Yaskawa INFORM job: X2_50&56B(90_180).JBI

/JOB
//NAME X2_50&56B(90_180)
//POS
///NPOS 378,378,378,17,0,0
///TOOL 0
///POSTYPE PULSE
///PULSE
C00000=-45487,-81749,-76140,-5313,88955,2714
C00001=-100725,-66680,-65098,-5325,101088,-31571
C00002=-135191,-12017,-32267,-15378,118169,-54834
C00003=-185881,43065,27917,-7885,118942,-78845
C00004=-185977,37643,25036,-7838,117929,-78810
C00005=-186017,35528,23980,-7818,117492,-78794
C00006=-186014,35949,26083,-7734,116424,-78717
C00007=-186017,35528,23980,-7818,117492,-78794
C00008=-187441,40927,31967,-8194,115230,-79185
C00009=-186781,38432,29365,-7969,115612,-78957
C00010=-187441,40927,31967,-8194,115230,-79185
C00011=-188109,40448,31416,-8451,115253,-79445
C00012=-188900,38382,29270,-8768,115424,-79764
C00013=-188109,40448,31416,-8451,115253,-79445
C00014=-187906,47991,35532,-8483,116603,-79469
C00015=-135191,-12017,-32267,-15378,118169,-54834
C00016=-100725,-66680,-65098,-5325,101088,-31571
C00017=-68653,-71679,-73408,-24733,95794,-85842
C00018=-66615,-75998,-75470,-24709,95531,-75346
C00019=-80537,-29900,-12555,-12207,96591,-80441
C00020=-81172,-32243,-10721,-12278,94215,-80425
C00021=-81559,-32147,-8308,-12330,92754,-80411
C00022=-81559,-31652,-7175,-12323,92320,-80369
C00023=-79890,-31226,-7999,-11978,93276,-79895
C00024=-78854,-29246,-5136,-11740,92696,-79487
C00025=-78019,-31526,-6644,-11553,92575,-79192
C00026=-78854,-29246,-5136,-11740,92696,-79487
C00027=-78535,-28461,-4244,-11667,92599,-79369
C00028=-79905,-29828,-5160,-11964,92267,-79802
C00029=-78535,-28461,-4244,-11667,92599,-79369
C00030=-80655,-29539,-12313,-12233,96610,-80484
C00031=-172905,9069,10368,-17661,103953,-63205
C00032=-172925,6453,11622,-17490,101927,-62911
C00033=-172953,5852,13232,-17402,100678,-62738
C00034=-172980,6410,14735,-17366,100062,-62659
C00035=-172934,5478,12205,-17429,101103,-62793
C00036=-174868,12262,20269,-17776,99277,-63224
C00037=-175653,10008,18253,-17959,99184,-63493
C00038=-174868,12262,20269,-17776,99277,-63224
C00039=-175466,10534,19114,-17901,98978,-63395
C00040=-174549,8650,17530,-17692,99183,-63095
C00041=-175466,10534,19114,-17901,98978,-63395
C00042=-175364,13912,17144,-18083,101810,-63784
C00043=-143557,-6058,-8183,-20909,99706,-63742
C00044=-116076,-21395,-35361,-8294,99864,41660
C00045=-116170,-16904,-19810,-8141,92666,42104
C00046=-120850,-15711,-13213,-8164,88779,40753
C00047=-120850,-15320,-11697,-8164,88052,40800
C00048=-120850,-15603,-12792,-8164,88575,40767
C00049=-118682,-15547,-12749,-8147,88797,41494
C00050=-118682,-15195,-11396,-8147,88151,41535
C00051=-119909,-15242,-11433,-8154,88024,41123
C00052=-118283,-15171,-11379,-8139,88193,41669
C00053=-118283,-17130,-20118,-8163,92522,41388
C00054=-123081,10517,-9626,-8350,99710,39267
C00055=-134850,49030,33201,-8140,92015,35751
C00056=-141062,59824,58615,-8076,81394,34310
C00057=-142218,64109,67353,-8122,78133,34125
C00058=-142677,66161,71300,-8151,76726,34060
C00059=-142679,67522,74254,-8187,75619,34134
C00060=-142677,66161,71300,-8151,76726,34060
C00061=-139671,63374,68885,-13312,76030,35539
C00062=-140369,64241,69903,-13301,75741,35326
C00063=-139671,63374,68885,-13312,76030,35539
C00064=-139134,61469,65218,-13265,77363,35582
C00065=-137783,55984,53040,-13137,82140,35542
C00066=-137153,72578,74728,-16498,89697,70863
C00067=-137090,72216,76874,-16484,88263,71078
C00068=-137090,73854,80265,-16487,87067,71239
C00069=-137090,73569,79683,-16486,87270,71212
C00070=-137224,70138,75519,-16503,88011,71066
C00071=-137093,72534,77607,-16485,87985,71116
C00072=-140530,75101,78865,-7193,89923,68947
C00073=-141437,70271,73879,-7337,90425,68614
C00074=-141815,70830,74551,-7395,90266,68496
C00075=-141437,68500,69903,-7348,91950,68525
C00076=-138489,28942,16401,-3523,91083,69516
C00077=-135724,-13299,-17509,-11404,84195,25469
C00078=-147110,-27573,-22260,-4915,65599,624
C00079=-144936,-25231,-14401,-13186,59518,1321
C00080=-144776,-24291,-13743,-13234,59620,1373
C00081=-145010,-25647,-14692,-13164,59472,1298
C00082=-145010,-26352,-16893,-13037,60439,1181
C00083=-144720,-24654,-15708,-13123,60625,1273
C00084=-144720,-24280,-14515,-13190,60096,1337
C00085=-145112,-27129,-17933,-12968,60658,1116
C00086=-149472,-33449,-22184,-828,57336,-10794
C00087=-149966,-29456,-16781,-629,56059,-10982
C00088=-150545,-29031,-16493,-385,56096,-11216
C00089=-149966,-29456,-16781,-629,56059,-10982
C00090=-143611,-50009,-41026,-3170,60566,-8561
C00091=-116233,-46088,-51369,-8218,97039,41795
C00092=-133480,-42531,-38521,-8139,89270,36398
C00093=-135471,-40868,-33851,-8115,87069,35859
C00094=-136262,-40121,-31922,-8108,86194,35645
C00095=-136263,-39693,-30384,-8112,85474,35691
C00096=-136262,-40121,-31922,-8108,86194,35645
C00097=-131087,-41226,-31195,-13244,85070,37562
C00098=-132294,-40915,-31003,-13224,84913,37159
C00099=-131087,-41226,-31195,-13244,85070,37562
C00100=-130160,-41921,-33014,-13249,85964,37789
C00101=-127831,-43444,-37404,-13266,88216,38359
C00102=-120126,-54973,-38990,-8175,84580,41274
C00103=-122393,-53255,-34311,-8216,82373,40644
C00104=-123299,-52483,-32378,-8234,81496,40391
C00105=-123299,-51827,-30705,-8247,80810,40437
C00106=-123299,-52483,-32378,-8234,81496,40391
C00107=-117579,-51909,-30953,-13332,81791,42614
C00108=-118939,-51968,-30986,-13356,81559,42167
C00109=-117579,-51909,-30953,-13332,81791,42614
C00110=-116541,-52550,-32737,-13293,82710,42875
C00111=-113955,-53926,-37043,-13200,85024,43525
C00112=-47420,-68852,-70475,-7734,99047,48455
C00113=-58856,-91847,-113443,-3781,117020,74641
C00114=-60236,-59653,-81414,-8514,109210,81552
C00115=-65712,-50088,-67931,-3279,110982,81026
C00116=-65935,-54727,-66929,-3231,107978,81030
C00117=-66231,-56054,-65409,-3227,106352,80970
C00118=-66421,-55660,-64438,-3238,105949,80915
C00119=-66309,-56041,-64890,-3229,106036,80952
C00120=-66048,-59202,-66118,-3188,105179,81066
C00121=-66309,-56041,-64890,-3229,106036,80952
C00122=-65984,-49861,-66477,-3286,110194,80952
C00123=-118683,-89548,-94864,6316,107762,74317
C00124=-118830,-94736,-93309,6169,104171,74077
C00125=-118897,-96147,-91968,6116,102635,73976
C00126=-118911,-94939,-90367,6104,102273,73953
C00127=-118926,-95247,-90740,6105,102345,73951
C00128=-120069,-98591,-91538,5957,101210,73497
C00129=-118926,-95247,-90740,6105,102345,73951
C00130=-124253,-93200,-90530,5582,103647,72150
C00131=-124297,-94887,-90828,5558,102970,72104
C00132=-122332,-96938,-91342,5745,102098,72750
C00133=-124297,-94887,-90828,5558,102970,72104
C00134=-123836,-88068,-93172,5765,107861,72497
C00135=-103947,-87224,-93768,-11726,103256,73456
C00136=-105491,-91629,-91965,-11598,99731,73257
C00137=-106242,-92046,-89539,-11549,97951,73163
C00138=-106280,-91630,-88956,-11545,97803,73164
C00139=-106194,-91849,-89665,-11554,98133,73164
C00140=-106981,-95473,-90615,-11530,96768,73018
C00141=-106194,-91849,-89665,-11554,98133,73164
C00142=-107390,-94613,-90436,-11549,97035,72851
C00143=-105229,-95826,-90624,-11481,96844,73620
C00144=-107390,-94613,-90436,-11549,97035,72851
C00145=-105129,-89034,-93253,-11689,101866,73178
C00146=-117235,-90812,-97794,-11932,101979,68958
C00147=-119184,-94938,-95823,-11777,98434,68628
C00148=-119997,-95229,-93380,-11717,96698,68512
C00149=-120000,-94762,-92745,-11713,96550,68526
C00150=-120085,-95315,-93448,-11717,96683,68484
C00151=-121254,-98780,-94295,-11676,95281,68213
C00152=-120085,-95315,-93448,-11717,96683,68484
C00153=-120732,-97303,-93959,-11694,95897,68335
C00154=-122720,-95241,-93443,-11703,96339,67606
C00155=-120732,-97303,-93959,-11694,95897,68335
C00156=-117928,-92127,-96991,-11873,100734,68840
C00157=-83815,-72409,-71600,-49856,101385,80874
C00158=-86977,-76307,-70966,-49554,98078,81004
C00159=-85918,-79626,-70912,-49280,97499,81857
C00160=-85722,-81512,-70616,-49126,96837,82303
C00161=-87678,-80975,-72090,-49364,96559,81447
C00162=-88529,-80279,-70734,-49348,95782,81419
C00163=-87018,-80378,-72384,-49396,97246,81423
C00164=-92255,-82689,-76075,-49623,95110,79856
C00165=-92255,-82357,-74554,-49552,94603,80124
C00166=-91886,-84274,-76762,-49584,95051,80076
C00167=-87038,-78982,-77882,-49995,99948,79968
C00168=-111885,-94745,-96836,-21175,93099,57761
C00169=-115356,-96241,-94167,-20812,89966,57066
C00170=-116782,-95898,-92034,-20669,88542,56800
C00171=-116805,-94979,-90810,-20667,88272,56838
C00172=-117687,-92490,-90484,-20584,89063,56388
C00173=-119638,-92586,-90524,-20383,88555,55777
C00174=-116782,-95072,-90979,-20669,88331,56836
C00175=-116675,-98914,-91892,-20684,87033,57096
C00176=-116782,-95072,-90979,-20669,88331,56836
C00177=-111949,-93327,-94846,-21154,92619,57823
C00178=-55380,-134082,-104834,-55812,75253,81172
C00179=-61753,-134169,-102482,-55825,70609,80463
C00180=-64815,-132350,-99998,-55791,68452,80067
C00181=-65073,-131468,-99170,-55790,68267,80036
C00182=-65012,-131683,-99347,-55795,68302,80050
C00183=-67421,-134585,-100123,-55949,66292,79958
C00184=-65012,-131683,-99347,-55795,68302,80050
C00185=-66833,-133758,-99865,-55902,66793,79972
C00186=-68699,-130981,-99713,-55278,66469,79035
C00187=-66833,-133758,-99865,-55902,66793,79972
C00188=-57706,-134492,-103408,-55942,73242,81128
C00189=-64785,-112873,-118243,-24954,102118,81978
C00190=-94326,-86621,-83484,35338,109503,87169
C00191=-91634,-91881,-83017,35113,105930,87131
C00192=-90294,-93871,-83332,35163,104694,87298
C00193=-90673,-91662,-79967,34941,104076,86932
C00194=-96279,-95614,-77654,39133,100534,74699
C00195=-97530,-94207,-78400,39125,102027,74707
C00196=-99906,-89889,-79610,39309,105429,74936
C00197=-93707,-90060,-101982,2678,109676,68403
C00198=-85859,-88563,-85007,-37375,108858,60120
C00199=-89767,-92929,-84612,-37372,105169,59726
C00200=-92261,-92553,-83552,-37602,103718,59151
C00201=-87809,-89294,-77804,-36664,104133,60948
C00202=-97825,-97090,-85633,-28728,98264,58810
C00203=-105101,-94972,-90460,-21721,102166,53461
C00204=-101619,-91841,-92201,-21697,105576,54126
C00205=-110011,-90138,-98551,-28023,73725,47627
C00206=-114073,-86949,-94757,-26595,71811,46539
C00207=-115644,-85550,-93357,-26007,71199,46082
C00208=-116827,-38850,-76508,-24575,105038,42322
C00209=-113194,-138803,-104651,-24561,74823,49786
C00210=-115995,-123992,-100550,-21546,88254,42562
C00211=-113813,-124047,-101616,-21486,89414,43150
C00212=-108993,-124666,-104884,-21332,92253,44397
C00213=-109211,-98340,-98499,-17204,97884,65653
C00214=-111963,-101539,-96259,-17038,94417,65168
C00215=-114319,-101452,-95162,-16976,93323,64488
C00216=-121130,-95827,-93982,-7505,98794,69297
C00217=-120137,-94785,-95042,-7509,100063,69562
C00218=-118600,-90390,-96949,-7580,103607,69872
C00219=-87744,-101201,-89183,-32285,100120,63549
C00220=-91822,-104522,-87796,-32421,96378,62986
C00221=-93007,-105888,-87219,-32449,95024,62902
C00222=-125171,-100001,-94421,-10746,96250,68519
C00223=-112189,-112791,-97117,-10082,92847,73286
C00224=-125737,-104595,-94231,-123,98676,80328
C00225=-125012,-83838,-85262,-564,111182,80520
C00226=-124880,-77934,-85992,-554,114665,80551
C00227=-118378,-61430,-80227,500,113656,60542
C00228=-119635,-65792,-78782,346,110532,60082
C00229=-120344,-67374,-78220,265,109375,59827
C00230=-117636,-69991,-79065,562,108539,60782
C00231=-61499,-79673,-75485,5801,99043,80116
C00232=-59682,-78713,-74784,5933,98973,80740
C00233=-58729,-76685,-75165,6027,100171,81128
C00234=-59096,-71470,-86943,6341,110071,81508
C00235=-60236,-59653,-81414,-8514,109210,81552
C00236=-58856,-91847,-113443,-3781,117020,74641
C00237=-47420,-68852,-70475,-7734,99047,48455
C00238=-126000,-95797,-97639,7032,71909,-3420
C00239=-125334,-73481,-62420,7403,61720,-3825
C00240=-136814,-5072,7481,-118,87452,-82611
C00241=-137691,-48649,-34753,-2434,90887,-80546
C00242=-137775,-50281,-31902,-2439,88294,-80524
C00243=-137810,-50839,-30689,-2442,87260,-80516
C00244=-135168,-51719,-31185,-2214,87179,-79626
C00245=-133081,-52293,-31505,-2034,87136,-78923
C00246=-130377,-52882,-31830,-1800,87108,-78013
C00247=-130424,-52342,-33062,-1804,88142,-78044
C00248=-109921,-30503,-12357,-16555,100596,-88828
C00249=-109696,-31149,-11049,-16422,99550,-88604
C00250=-109235,-30430,-9939,-16278,99338,-88414
C00251=-108888,-29584,-8170,-16145,98777,-88217
C00252=-108084,-28000,-11018,-16080,101404,-88284
C00253=-146524,-12798,-32,1632,107432,-69723
C00254=-145636,-15796,-268,1931,106019,-69429
C00255=-148965,-15940,435,4110,105287,-67260
C00256=-149102,-15441,1522,4054,104879,-67319
C00257=-149548,-12799,1040,3936,106552,-67422
C00258=-137932,-46455,-34045,-2456,91570,-80642
C00259=-130584,-47998,-33152,-21701,103265,-82699
C00260=-131924,-51228,-32028,-21814,100720,-82725
C00261=-132035,-52540,-31560,-21763,99795,-82595
C00262=-133096,-52283,-31444,-22032,99580,-82945
C00263=-135164,-51769,-31262,-22544,99165,-83631
C00264=-135522,-51681,-31234,-22630,99088,-83749
C00265=-135156,-50442,-31749,-22619,100068,-83801
C00266=-145953,-54402,-37679,-17502,96627,-81619
C00267=-150690,-47590,-28968,-15173,97194,-77528
C00268=-141688,-67515,-39498,-21463,83995,-90539
C00269=-138380,-68197,-47605,-21119,89179,-90269
C00270=-135468,-61779,-51499,-19715,96090,-83313
C00271=-146504,11659,2252,-17659,107540,-74925
C00272=-144153,-20650,-13732,-15502,93070,1402
C00273=-144800,-23297,881,-19511,75808,35743
C00274=-150190,-18698,6871,-14781,74684,33485
C00275=-147156,-18843,9866,-19821,72199,35502
C00276=-149144,-27907,3634,-19922,70959,34997
C00277=-146448,7715,36431,-22348,89479,40067
C00278=-145889,24730,54854,-22060,94685,42086
C00279=-143819,24834,51946,-21414,96917,42392
C00280=-152079,-13657,11289,-11329,66320,30599
C00281=-154288,-10621,16286,-8724,64794,29674
C00282=-151904,106,24911,-8978,65250,30498
C00283=-150907,-2622,20158,-8985,66862,30731
C00284=-148148,-14759,14441,-17311,62501,33163
C00285=-153240,-11311,16162,-10073,64214,30249
C00286=-151074,-2242,23117,-10293,64850,30978
C00287=-150611,-3939,19670,-10247,66139,31030
C00288=-148132,-4021,18992,-11949,66408,32059
C00289=-147374,-3194,21269,-13667,65169,32648
C00290=-146197,4054,27436,-13805,65293,33065
C00291=-152653,-4647,20265,-5226,59206,14792
C00292=-154418,-25114,11432,-1101,38258,22446
C00293=-154596,-31771,2822,-953,40134,22334
C00294=-135242,-54877,-19518,-11584,43472,31405
C00295=-131236,-19596,-17600,-13529,71052,30429
C00296=-140706,-23702,-4175,-12836,48543,13474
C00297=-139806,-19028,764,-13410,48067,13944
C00298=-142658,-11173,6654,-18063,50404,18129
C00299=-141158,-15186,3600,-18761,50563,18771
C00300=-142435,-9097,12555,-18853,48016,18701
C00301=-142049,-7157,14085,-20669,49065,20425
C00302=-142257,-9387,11148,-20387,49635,20204
C00303=-144365,-13616,3568,-3735,54240,8270
C00304=-145823,-13393,6250,-1324,50480,7579
C00305=-145532,-11229,7851,-5107,50939,11169
C00306=-140850,-20387,-3678,-6927,53662,12969
C00307=-124087,52798,66602,-30516,90034,63653
C00308=-125471,40650,54753,-32699,86509,59979
C00309=-125334,44720,63004,-32764,84027,60751
C00310=-121896,62283,77480,-32170,85396,61678
C00311=-136105,75569,91402,-14378,82982,62392
C00312=-137341,77557,93952,-14596,82241,62066
C00313=-141168,85934,104737,-15299,79317,61146
C00314=-141539,87094,106260,-15375,78917,61072
C00315=-141741,86606,105619,-15400,79023,60993
C00316=-141171,84118,98448,-15196,82155,60793
C00317=-132001,54931,46945,-19188,86263,30068
C00318=-132148,77644,76370,-19381,80137,30989
C00319=-133367,86129,89618,-16102,76593,30820
C00320=-134153,81899,83498,-14098,78199,30187
C00321=-134623,67905,67625,-12481,69763,30818
C00322=-134986,36263,31606,-9687,63888,24183
C00323=-134666,27103,16729,-9479,68314,23935
C00324=-130420,39472,29702,-18859,92900,38190
C00325=-131547,40725,34135,-18850,90663,38133
C00326=-134032,43651,38469,-15292,90000,37322
C00327=-134717,31522,25950,-15335,91293,36921
C00328=-133273,44284,38720,-16717,93907,38368
C00329=-131769,55424,45596,-17778,98765,39318
C00330=-127656,48680,32292,-16283,104912,42086
C00331=-116663,7338,4481,-17873,88938,41861
C00332=-82713,25471,38030,-41323,96034,53690
C00333=-86390,18515,43854,-41800,88900,54935
C00334=-85131,26101,60384,-49314,87065,55858
C00335=-88537,53193,89669,-50569,82685,56609
C00336=-87361,53333,88208,-50128,83897,56499
C00337=-87606,32039,49279,-49923,92343,51642
C00338=-120401,-109118,-96895,-24846,84275,3219
C00339=-171543,-75667,-77525,32488,107850,-47798
C00340=-132158,4506,-3799,21442,87877,-38180
C00341=-135903,57798,67571,35925,99624,-57782
C00342=-135834,61045,74411,35664,97518,-58450
C00343=-136852,65101,79345,35223,97458,-58869
C00344=-135824,2781,6571,30163,84476,-36889
C00345=-132310,1940,5711,27060,83090,-36079
C00346=-131484,15794,17971,27055,82441,-35917
C00347=-137267,10911,1717,27131,91031,-36122
C00348=-146203,-27363,-23504,26744,90214,-39705
C00349=-126939,-13199,-3011,17863,102554,-59788
C00350=-123418,-15871,2353,18433,97326,-59310
C00351=-121180,-11626,8848,18695,97500,-62472
C00352=-121861,-10835,10563,18474,97032,-62783
C00353=-122570,-10261,12471,18233,96354,-63137
C00354=-117580,-17478,3718,13074,93264,-62869
C00355=-122301,-18046,-869,17501,95215,-65467
C00356=-137808,-17234,-5965,14129,101643,-70132
C00357=-160865,-72571,-62696,26432,95765,-43985
C00358=-33343,-40499,-55087,-21473,103101,-25780
C00359=-34531,-11607,-34091,-29923,106513,-58273
C00360=-34985,-14035,-31998,-29527,104140,-57811
C00361=-34859,-13066,-29764,-29400,103418,-57570
C00362=-36609,-20544,-36296,-27578,100646,-57392
C00363=-52934,-69115,-66821,-23349,86237,-60131
C00364=-53727,-71032,-72534,-20342,85587,-60124
C00365=-146487,-18846,-10598,-19725,94468,-68028
C00366=-155890,-2777,10204,-12003,101739,-63000
C00367=-156750,-807,13372,-12200,100693,-63202
C00368=-157443,816,16029,-12357,99805,-63356
C00369=-157211,1579,14506,-12356,101141,-63409
C00370=-145375,-16597,89,-21780,91791,-76946
C00371=-153197,-12711,3322,-13630,93085,-80939
C00372=-151754,-15041,1558,-14681,91924,-82917
C00373=-145475,-7318,12723,-24819,92922,-88907
C00374=-142776,-6009,11285,-24301,95132,-88379
C00375=-137963,-3619,4000,-23654,101759,-87941
C00376=-103503,-37411,-26995,-22689,104461,-77175
C00377=2000,-113393,-91320,0,88983,0
BC00000=213492,669309,586749
BC00001=279836,668491,248946
BC00002=347085,719558,248946
BC00003=397217,757626,248946
BC00004=397217,757626,248946
BC00005=397217,757626,248946
BC00006=397217,757626,248946
BC00007=397217,757626,248946
BC00008=397217,757626,248946
BC00009=397217,757626,248946
BC00010=397217,757626,248946
BC00011=397217,757626,248946
BC00012=397217,757626,248946
BC00013=397217,757626,248946
BC00014=397217,757626,248946
BC00015=347085,719558,248946
BC00016=279836,668491,248946
BC00017=74259,666735,420956
BC00018=74259,755070,420956
BC00019=74259,755070,420956
BC00020=74259,755070,420956
BC00021=74259,755070,420956
BC00022=74259,755070,420956
BC00023=74259,755070,420956
BC00024=74259,755070,420956
BC00025=74259,755070,420956
BC00026=74259,755070,420956
BC00027=74259,755070,420956
BC00028=74259,755070,420956
BC00029=74259,755070,420956
BC00030=74259,755070,420956
BC00031=168853,756619,369390
BC00032=168853,756619,369390
BC00033=168853,756619,369390
BC00034=168853,756619,369390
BC00035=168853,756619,369390
BC00036=168853,756619,369390
BC00037=168853,756619,369390
BC00038=168853,756619,369390
BC00039=168853,756619,369390
BC00040=168853,756619,369390
BC00041=168853,756619,369390
BC00042=168853,756619,369390
BC00043=153069,767391,383312
BC00044=133900,791089,347452
BC00045=133902,791088,347446
BC00046=133902,791088,347446
BC00047=133902,791088,347446
BC00048=133902,791088,347446
BC00049=133902,791088,347446
BC00050=133902,791088,347446
BC00051=133902,791088,347446
BC00052=133902,791088,347446
BC00053=133902,791088,347446
BC00054=133900,791089,347452
BC00055=133900,791089,347452
BC00056=133900,791089,347452
BC00057=133900,791089,347452
BC00058=133900,791089,347452
BC00059=133900,791089,347452
BC00060=133900,791089,347452
BC00061=133900,791089,347452
BC00062=133900,791089,347452
BC00063=133900,791089,347452
BC00064=133900,791089,347452
BC00065=133900,791089,347452
BC00066=133900,791089,347451
BC00067=133900,791089,347451
BC00068=133900,791089,347451
BC00069=133900,791089,347451
BC00070=133900,791089,347451
BC00071=133900,791089,347451
BC00072=133900,791089,347451
BC00073=133900,791089,347451
BC00074=133900,791089,347451
BC00075=133900,791089,347451
BC00076=133900,791089,347451
BC00077=133900,791089,347451
BC00078=133899,791089,347449
BC00079=133899,791089,347449
BC00080=133899,791089,347449
BC00081=133899,791089,347449
BC00082=133899,791089,347449
BC00083=133899,791089,347449
BC00084=133899,791089,347449
BC00085=133899,791089,347449
BC00086=133899,791089,347449
BC00087=133899,791089,347449
BC00088=133899,791089,347449
BC00089=133899,791089,347449
BC00090=133899,791089,347449
BC00091=91689,791089,305907
BC00092=91689,791089,305907
BC00093=91689,791089,305907
BC00094=91689,791089,305907
BC00095=91689,791089,305907
BC00096=91689,791089,305907
BC00097=91689,791089,305907
BC00098=91689,791089,305907
BC00099=91689,791089,305907
BC00100=91689,791089,305907
BC00101=91689,791089,305907
BC00102=65725,737951,350532
BC00103=65725,737951,350532
BC00104=65725,737951,350532
BC00105=65725,737951,350532
BC00106=65725,737951,350532
BC00107=65725,737951,350532
BC00108=65725,737951,350532
BC00109=65725,737951,350532
BC00110=65725,737951,350532
BC00111=65725,737951,350532
BC00112=45615,670175,524343
BC00113=269563,738996,1075229
BC00114=398174,782420,1075175
BC00115=398174,782420,1075175
BC00116=398174,782420,1075175
BC00117=398174,782420,1075175
BC00118=398174,782420,1075175
BC00119=398174,782420,1075175
BC00120=398174,782420,1075175
BC00121=398174,782420,1075175
BC00122=398174,782420,1075175
BC00123=387355,830302,1075175
BC00124=387355,830302,1075175
BC00125=387355,830302,1075175
BC00126=387355,830302,1075175
BC00127=387355,830302,1075175
BC00128=387355,830302,1075175
BC00129=387355,830302,1075175
BC00130=387355,830302,1075175
BC00131=387355,830302,1075175
BC00132=387355,830302,1075175
BC00133=387355,830302,1075175
BC00134=387355,830302,1075175
BC00135=398174,816751,1075175
BC00136=398174,816751,1075175
BC00137=398174,816751,1075175
BC00138=398174,816751,1075175
BC00139=398174,816751,1075175
BC00140=398174,816751,1075175
BC00141=398174,816751,1075175
BC00142=398174,816751,1075175
BC00143=398174,816751,1075175
BC00144=398174,816751,1075175
BC00145=398174,816751,1075175
BC00146=394174,829691,1075175
BC00147=394174,829691,1075175
BC00148=394174,829691,1075175
BC00149=394174,829691,1075175
BC00150=394174,829691,1075175
BC00151=394174,829691,1075175
BC00152=394174,829691,1075175
BC00153=394174,829691,1075175
BC00154=394174,829691,1075175
BC00155=394174,829691,1075175
BC00156=394174,829691,1075175
BC00157=398174,810220,1075175
BC00158=398174,810220,1075175
BC00159=398174,810220,1075175
BC00160=398174,810220,1075175
BC00161=398174,810220,1075175
BC00162=398174,810220,1075175
BC00163=398174,810220,1075175
BC00164=398174,810220,1075175
BC00165=398174,810220,1075175
BC00166=398174,810220,1075175
BC00167=398174,810220,1075175
BC00168=398174,820048,1075175
BC00169=398174,820048,1075175
BC00170=398174,820048,1075175
BC00171=398174,820048,1075175
BC00172=398174,820048,1075175
BC00173=398174,820048,1075175
BC00174=398174,820048,1075175
BC00175=398174,820048,1075175
BC00176=398174,820048,1075175
BC00177=398174,820048,1075175
BC00178=357533,882194,1075175
BC00179=357533,882194,1075175
BC00180=357533,882194,1075175
BC00181=357533,882194,1075175
BC00182=357533,882194,1075175
BC00183=357533,882194,1075175
BC00184=357533,882194,1075175
BC00185=357533,882194,1075175
BC00186=357533,882194,1075175
BC00187=357533,882194,1075175
BC00188=357533,882194,1075175
BC00189=340885,876696,1075175
BC00190=309760,866417,1075175
BC00191=309760,866417,1075175
BC00192=309760,866417,1075175
BC00193=309760,866417,1075175
BC00194=309760,866417,1075175
BC00195=309760,866417,1075175
BC00196=309760,866417,1075175
BC00197=346143,852026,1075175
BC00198=394169,833030,1075175
BC00199=394169,833030,1075175
BC00200=394169,833030,1075175
BC00201=394169,833030,1075175
BC00202=394169,833030,1075175
BC00203=394169,833030,1075175
BC00204=394169,833030,1075175
BC00205=398174,851161,1075175
BC00206=398174,851161,1075175
BC00207=398174,851161,1075175
BC00208=398174,851161,1075175
BC00209=398174,851161,1075175
BC00210=398174,851161,1075175
BC00211=398174,851161,1075175
BC00212=398174,851161,1075175
BC00213=383646,835540,1075175
BC00214=383646,835540,1075175
BC00215=383647,835541,1075174
BC00216=383646,835540,1075175
BC00217=383646,835540,1075175
BC00218=383646,835540,1075175
BC00219=398174,834635,1075175
BC00220=398174,834635,1075175
BC00221=398174,834635,1075175
BC00222=398174,834635,1075175
BC00223=398174,834635,1075175
BC00224=398174,834635,1075175
BC00225=398174,834635,1075175
BC00226=398174,834635,1075175
BC00227=398174,805809,1075175
BC00228=398174,805809,1075175
BC00229=398174,805809,1075175
BC00230=398174,805809,1075175
BC00231=398174,805809,1075175
BC00232=398174,805809,1075175
BC00233=398174,805809,1075175
BC00234=398174,805809,1075175
BC00235=398174,782420,1075175
BC00236=269563,738996,1075229
BC00237=45615,670175,524343
BC00238=94279,678895,315353
BC00239=94279,729713,315353
BC00240=135603,767285,503004
BC00241=127958,749365,374153
BC00242=127958,749365,374153
BC00243=127958,749365,374153
BC00244=127958,749365,374153
BC00245=127958,749365,374153
BC00246=127958,749365,374153
BC00247=127958,749365,374153
BC00248=127958,749365,374153
BC00249=127958,749365,374153
BC00250=127958,749365,374153
BC00251=127958,749365,374153
BC00252=127958,749365,374153
BC00253=127958,749365,374153
BC00254=127958,749365,374153
BC00255=127958,749365,374153
BC00256=127958,749365,374153
BC00257=127958,749365,374153
BC00258=127958,749365,374153
BC00259=104823,777232,320967
BC00260=104823,777232,320967
BC00261=104823,777232,320967
BC00262=104823,777232,320967
BC00263=104823,777232,320967
BC00264=104823,777232,320967
BC00265=104823,777232,320967
BC00266=104823,777232,320967
BC00267=104823,777232,320967
BC00268=104823,777232,320967
BC00269=104823,777232,320967
BC00270=104823,777232,320967
BC00271=148105,732999,367459
BC00272=136799,735677,423222
BC00273=131883,736842,447466
BC00274=131883,736842,447466
BC00275=131883,736842,447466
BC00276=131883,736842,447466
BC00277=131883,736842,447466
BC00278=131883,736842,447466
BC00279=131883,736842,447466
BC00280=135864,729332,463750
BC00281=135864,729332,463750
BC00282=135864,729332,463750
BC00283=135864,729332,463750
BC00284=135957,757580,463073
BC00285=135957,757580,463073
BC00286=135957,757580,463073
BC00287=135957,757580,463073
BC00288=132965,771777,450481
BC00289=132965,771777,450481
BC00290=132965,771777,450481
BC00291=132965,771777,450481
BC00292=132965,771777,450481
BC00293=132965,771777,450481
BC00294=132965,771777,450481
BC00295=129716,779092,399778
BC00296=129716,779092,399778
BC00297=129716,779092,399778
BC00298=129716,779092,399778
BC00299=129716,779092,399778
BC00300=129716,779092,399778
BC00301=129716,779092,399778
BC00302=129716,779092,399778
BC00303=129716,779092,399778
BC00304=129716,779092,399778
BC00305=129716,779092,399778
BC00306=129716,779092,399778
BC00307=129716,795131,399778
BC00308=129716,795131,399778
BC00309=129716,795131,399778
BC00310=129716,795131,399778
BC00311=129716,795131,399778
BC00312=129716,795131,399778
BC00313=129716,795131,399778
BC00314=129716,795131,399778
BC00315=129716,795131,399778
BC00316=129716,795131,399778
BC00317=124387,791089,316625
BC00318=124387,789553,316625
BC00319=119293,789553,296084
BC00320=117256,789553,287867
BC00321=117256,789553,287867
BC00322=112196,789553,268708
BC00323=112196,789553,268708
BC00324=113936,791089,281332
BC00325=113936,791089,281332
BC00326=113936,791089,281332
BC00327=113936,791089,281332
BC00328=113936,791089,281332
BC00329=113936,791089,281332
BC00330=113936,791089,281332
BC00331=116869,773103,397669
BC00332=116869,773103,397669
BC00333=116869,773103,397669
BC00334=116869,773103,397669
BC00335=116869,773103,397669
BC00336=116869,773103,397669
BC00337=116996,772325,398387
BC00338=133980,668182,494562
BC00339=6392,668182,323571
BC00340=6392,776369,323571
BC00341=6392,786149,323571
BC00342=6392,786149,323571
BC00343=6392,786149,323571
BC00344=6392,786149,323571
BC00345=6392,786149,323571
BC00346=6392,786149,323571
BC00347=6392,786149,323571
BC00348=6392,734041,397800
BC00349=6392,734041,397800
BC00350=6392,734041,397800
BC00351=5812,733225,400788
BC00352=6392,733053,399870
BC00353=6392,734041,402294
BC00354=6392,734041,399183
BC00355=6392,734041,397800
BC00356=6392,734041,397800
BC00357=6392,674729,482291
BC00358=159586,688686,294802
BC00359=173113,745279,189268
BC00360=173113,745279,189268
BC00361=173113,745279,189268
BC00362=173113,745279,189268
BC00363=173113,745279,189268
BC00364=173113,745279,189268
BC00365=329544,744159,387532
BC00366=329544,744159,387532
BC00367=329544,744159,387532
BC00368=329544,744159,387532
BC00369=329544,744159,387532
BC00370=329544,744159,387532
BC00371=329544,744159,387532
BC00372=329544,744159,387532
BC00373=329544,744159,387532
BC00374=329544,744159,387532
BC00375=329544,744159,387532
BC00376=296372,673105,416449
BC00377=87189,666204,1075229
EC00000=798156,1112951
EC00001=798156,1112951
EC00002=798156,1112951
EC00003=798156,1112951
EC00004=798156,1112951
EC00005=798156,1112951
EC00006=798156,1112951
EC00007=798156,1112951
EC00008=798156,1112951
EC00009=798156,1112951
EC00010=798156,1112951
EC00011=798156,1112951
EC00012=798156,1112951
EC00013=798156,1112951
EC00014=798156,1112951
EC00015=798156,1112951
EC00016=798156,1112951
EC00017=798156,1112951
EC00018=798156,1112951
EC00019=798156,1112951
EC00020=798156,1112951
EC00021=798156,1112951
EC00022=798156,1112951
EC00023=798156,1112951
EC00024=798156,1112951
EC00025=798156,1112951
EC00026=798156,1112951
EC00027=798156,1112951
EC00028=798156,1112951
EC00029=798156,1112951
EC00030=798156,1112951
EC00031=798156,1112951
EC00032=798156,1112951
EC00033=798156,1112951
EC00034=798156,1112951
EC00035=798156,1112951
EC00036=798156,1112951
EC00037=798156,1112951
EC00038=798156,1112951
EC00039=798156,1112951
EC00040=798156,1112951
EC00041=798156,1112951
EC00042=798156,1112951
EC00043=798156,1112951
EC00044=798156,1112951
EC00045=798154,1112949
EC00046=798154,1112949
EC00047=798154,1112949
EC00048=798154,1112949
EC00049=798154,1112949
EC00050=798154,1112949
EC00051=798154,1112949
EC00052=798154,1112949
EC00053=798154,1112949
EC00054=798156,1112951
EC00055=798156,1112951
EC00056=798156,1112951
EC00057=798156,1112951
EC00058=798156,1112951
EC00059=798156,1112951
EC00060=798156,1112951
EC00061=798156,1112951
EC00062=798156,1112951
EC00063=798156,1112951
EC00064=798156,1112951
EC00065=798156,1112951
EC00066=798155,1112949
EC00067=798155,1112949
EC00068=798155,1112949
EC00069=798155,1112949
EC00070=798155,1112949
EC00071=798155,1112949
EC00072=798155,1112949
EC00073=798155,1112949
EC00074=798155,1112949
EC00075=798155,1112949
EC00076=798155,1112949
EC00077=798155,1112949
EC00078=798154,1112948
EC00079=798154,1112948
EC00080=798154,1112948
EC00081=798154,1112948
EC00082=798154,1112948
EC00083=798154,1112948
EC00084=798154,1112948
EC00085=798154,1112948
EC00086=798154,1112948
EC00087=798154,1112948
EC00088=798154,1112948
EC00089=798154,1112948
EC00090=798154,1112948
EC00091=798156,1112951
EC00092=798156,1112951
EC00093=798156,1112951
EC00094=798156,1112951
EC00095=798156,1112951
EC00096=798156,1112951
EC00097=798156,1112951
EC00098=798156,1112951
EC00099=798156,1112951
EC00100=798156,1112951
EC00101=798156,1112951
EC00102=798156,1112951
EC00103=798156,1112951
EC00104=798156,1112951
EC00105=798156,1112951
EC00106=798156,1112951
EC00107=798156,1112951
EC00108=798156,1112951
EC00109=798156,1112951
EC00110=798156,1112951
EC00111=798156,1112951
EC00112=798156,1112951
EC00113=906908,1112951
EC00114=975524,1112951
EC00115=975524,1112951
EC00116=975524,1112951
EC00117=975524,1112951
EC00118=975524,1112951
EC00119=975524,1112951
EC00120=975524,1112951
EC00121=975524,1112951
EC00122=975524,1112951
EC00123=975524,1112951
EC00124=975524,1112951
EC00125=975524,1112951
EC00126=975524,1112951
EC00127=975524,1112951
EC00128=975524,1112951
EC00129=975524,1112951
EC00130=975524,1112951
EC00131=975524,1112951
EC00132=975524,1112951
EC00133=975524,1112951
EC00134=975524,1112951
EC00135=975524,1112951
EC00136=975524,1112951
EC00137=975524,1112951
EC00138=975524,1112951
EC00139=975524,1112951
EC00140=975524,1112951
EC00141=975524,1112951
EC00142=975524,1112951
EC00143=975524,1112951
EC00144=975524,1112951
EC00145=975524,1112951
EC00146=975524,1112951
EC00147=975524,1112951
EC00148=975524,1112951
EC00149=975524,1112951
EC00150=975524,1112951
EC00151=975524,1112951
EC00152=975524,1112951
EC00153=975524,1112951
EC00154=975524,1112951
EC00155=975524,1112951
EC00156=975524,1112951
EC00157=975524,1112951
EC00158=975524,1112951
EC00159=975524,1112951
EC00160=975524,1112951
EC00161=975524,1112951
EC00162=975524,1112951
EC00163=975524,1112951
EC00164=975524,1112951
EC00165=975524,1112951
EC00166=975524,1112951
EC00167=975524,1112951
EC00168=975524,1112951
EC00169=975524,1112951
EC00170=975524,1112951
EC00171=975524,1112951
EC00172=975524,1112951
EC00173=975524,1112951
EC00174=975524,1112951
EC00175=975524,1112951
EC00176=975524,1112951
EC00177=975524,1112951
EC00178=975524,1112951
EC00179=975524,1112951
EC00180=975524,1112951
EC00181=975524,1112951
EC00182=975524,1112951
EC00183=975524,1112951
EC00184=975524,1112951
EC00185=975524,1112951
EC00186=975524,1112951
EC00187=975524,1112951
EC00188=975524,1112951
EC00189=975524,1112951
EC00190=975524,1112951
EC00191=975524,1112951
EC00192=975524,1112951
EC00193=975524,1112951
EC00194=975524,1112951
EC00195=975524,1112951
EC00196=975524,1112951
EC00197=975524,1112951
EC00198=975524,1112951
EC00199=975524,1112951
EC00200=975524,1112951
EC00201=975524,1112951
EC00202=975524,1112951
EC00203=975524,1112951
EC00204=975524,1112951
EC00205=975524,1112951
EC00206=975524,1112951
EC00207=975524,1112951
EC00208=975524,1112951
EC00209=975524,1112951
EC00210=975524,1112951
EC00211=975524,1112951
EC00212=975524,1112951
EC00213=975524,1112951
EC00214=975524,1112951
EC00215=975522,1112950
EC00216=975524,1112951
EC00217=975524,1112951
EC00218=975524,1112951
EC00219=975524,1112951
EC00220=975524,1112951
EC00221=975524,1112951
EC00222=975524,1112951
EC00223=975524,1112951
EC00224=975524,1112951
EC00225=975524,1112951
EC00226=975524,1112951
EC00227=975524,1112951
EC00228=975524,1112951
EC00229=975524,1112951
EC00230=975524,1112951
EC00231=975524,1112951
EC00232=975524,1112951
EC00233=975524,1112951
EC00234=975524,1112951
EC00235=975524,1112951
EC00236=906908,1112951
EC00237=798156,1112951
EC00238=798156,1112951
EC00239=798156,1112951
EC00240=798156,1112951
EC00241=798156,1112951
EC00242=798156,1112951
EC00243=798156,1112951
EC00244=798156,1112951
EC00245=798156,1112951
EC00246=798156,1112951
EC00247=798156,1112951
EC00248=798156,1112951
EC00249=798156,1112951
EC00250=798156,1112951
EC00251=798156,1112951
EC00252=798156,1112951
EC00253=798156,1112951
EC00254=798156,1112951
EC00255=798156,1112951
EC00256=798156,1112951
EC00257=798156,1112951
EC00258=798156,1112951
EC00259=798156,1112951
EC00260=798156,1112951
EC00261=798156,1112951
EC00262=798156,1112951
EC00263=798156,1112951
EC00264=798156,1112951
EC00265=798156,1112951
EC00266=798156,1112951
EC00267=798156,1112951
EC00268=798156,1112951
EC00269=798156,1112951
EC00270=798156,1112951
EC00271=798156,1112951
EC00272=798156,1112951
EC00273=798156,1112951
EC00274=798156,1112951
EC00275=798156,1112951
EC00276=798156,1112951
EC00277=798156,1112951
EC00278=798156,1112951
EC00279=798156,1112951
EC00280=798156,1112951
EC00281=798156,1112951
EC00282=798156,1112951
EC00283=798156,1112951
EC00284=798156,1112951
EC00285=798156,1112951
EC00286=798156,1112951
EC00287=798156,1112951
EC00288=798156,1112951
EC00289=798156,1112951
EC00290=798156,1112951
EC00291=798156,1112951
EC00292=798156,1112951
EC00293=798156,1112951
EC00294=798156,1112951
EC00295=798156,1112951
EC00296=798156,1112951
EC00297=798156,1112951
EC00298=798156,1112951
EC00299=798156,1112951
EC00300=798156,1112951
EC00301=798156,1112951
EC00302=798156,1112951
EC00303=798156,1112951
EC00304=798156,1112951
EC00305=798156,1112951
EC00306=798156,1112951
EC00307=798156,1112951
EC00308=798156,1112951
EC00309=798156,1112951
EC00310=798156,1112951
EC00311=798156,1112951
EC00312=798156,1112951
EC00313=798156,1112951
EC00314=798156,1112951
EC00315=798156,1112951
EC00316=798156,1112951
EC00317=798156,1112951
EC00318=798156,1112951
EC00319=798156,1112951
EC00320=798156,1112951
EC00321=798156,1112951
EC00322=798156,1112951
EC00323=798156,1112951
EC00324=798156,1112951
EC00325=798156,1112951
EC00326=798156,1112951
EC00327=798156,1112951
EC00328=798156,1112951
EC00329=798156,1112951
EC00330=798156,1112951
EC00331=798156,1112951
EC00332=798156,1112951
EC00333=798156,1112951
EC00334=798156,1112951
EC00335=798156,1112951
EC00336=798156,1112951
EC00337=798156,1112951
EC00338=798156,1112951
EC00339=798156,1112951
EC00340=798156,1112951
EC00341=798156,1112951
EC00342=798156,1112951
EC00343=798156,1112951
EC00344=798156,1112951
EC00345=798156,1112951
EC00346=798156,1112951
EC00347=798156,1112951
EC00348=798156,1112951
EC00349=798156,1112951
EC00350=798156,1112951
EC00351=798156,1112951
EC00352=798156,1112951
EC00353=798156,1112951
EC00354=798156,1112951
EC00355=798156,1112951
EC00356=798156,1112951
EC00357=798156,1112951
EC00358=798156,1112951
EC00359=798156,1112951
EC00360=798156,1112951
EC00361=798156,1112951
EC00362=798156,1112951
EC00363=798156,1112951
EC00364=798156,1112951
EC00365=798156,1112951
EC00366=798156,1112951
EC00367=798156,1112951
EC00368=798156,1112951
EC00369=798156,1112951
EC00370=798156,1112951
EC00371=798156,1112951
EC00372=798156,1112951
EC00373=798156,1112951
EC00374=798156,1112951
EC00375=798156,1112951
EC00376=798156,1112951
EC00377=798156,1112951
///POSTYPE BASE
///RECTAN
///RCONF 0,0,0,0,0,0,0,0,0,0,0,0,0,0,0,0,0,0,0,0,0,0,0,0
P00006=0.222,-3.123,-1.508,0.0000,0.0000,0.0000
P00021=-0.225,-6.128,-0.405,0.0000,0.0000,0.0000
P00022=0.222,-3.123,-1.508,0.0000,0.0000,0.0000
P00023=0.143,-0.036,0.682,0.0000,0.0000,0.0000
P00024=0.145,-0.552,1.326,0.0000,0.0000,0.0000
P00025=-2.003,0.006,0.728,0.0000,0.0000,0.0000
P00026=0.562,-0.002,-0.337,0.0000,0.0000,0.0000
P00027=-0.746,0.015,-9.096,0.0000,0.0000,0.0000
P00028=-2.237,-0.018,-7.702,0.0000,0.0000,0.0000
P00029=-2.156,-0.086,-4.681,0.0000,0.0000,0.0000
P00032=1.957,0.503,-7.217,0.0000,0.0000,0.0000
///RCONF 0,0,0,0,1,0,0,0,0,0,0,0,0,0,0,0,0,0,0,0,0,0,0,0
P00033=-0.123,0.612,-5.012,0.0000,0.0000,0.0000
///RCONF 0,0,0,0,0,0,0,0,0,0,0,0,0,0,0,0,0,0,0,0,0,0,0,0
P00034=-0.304,0.773,-2.693,0.0000,0.0000,0.0000
P00050=4.296,-4.501,-0.826,0.0000,0.0000,0.0000
P00051=0.367,3.892,0.009,0.0000,0.0000,0.0000
P00063=0.036,-0.654,-3.005,0.0000,0.0000,0.0000
P00099=-0.837,6.343,-3.499,0.0000,0.0000,0.0000
//INST
///DATE 2024/11/05 10:16
///ATTR SC,RW
///GROUP1 RB1,BS1
///GROUP2 ST1
NOP
'X2_50&56B(90_180)
'Down
MOVJ C00000 BC00000 VJ=100.00  +MOVJ EC00000 VJ=100.00
MOVJ C00001 BC00001 VJ=100.00  +MOVJ EC00001 VJ=100.00
MOVJ C00002 BC00002 VJ=100.00  +MOVJ EC00002 VJ=100.00
'Path S4514
SFTOF3D
MOVJ C00003 BC00003 VJ=100.00  +MOVJ EC00003 VJ=100.00
MOVL C00004 BC00004 V=800.0  +MOVJ EC00004 VJ=100.00
SMOVL C00005 BC00005 V=166.7  +MOVJ EC00005
SREFP 3 C00006 BC00006  +REFP EC00006
CALL JOB:SEARCH-R1-S13D
SET P034 P006
SFTON3D P034
SMOVL C00007 BC00007 V=166.7  +MOVJ EC00007
SMOVL C00008 BC00008 V=166.7  +MOVJ EC00008
SREFP 3 C00009 BC00009  +REFP EC00009
CALL JOB:SEARCH-R1-S13D
SET P034 P006
SFTON3D P034
SMOVL C00010 BC00010 V=166.7  +MOVJ EC00010
SMOVL C00011 BC00011 V=166.7  +MOVJ EC00011
SREFP 3 C00012 BC00012  +REFP EC00012
CALL JOB:SEARCH-R1-S13D
SET P034 P006
SFTON3D P034
SMOVL C00013 BC00013 V=166.7  +MOVJ EC00013
MOVL C00014 BC00014 V=1000.0  +MOVJ EC00014 VJ=100.00
'EndPath S4514
MOVJ C00015 BC00015 VJ=100.00  +MOVJ EC00015 VJ=100.00
MOVJ C00016 BC00016 VJ=100.00  +MOVJ EC00016 VJ=100.00
MOVJ C00017 BC00017 VJ=100.00  +MOVJ EC00017 VJ=100.00
MOVJ C00018 BC00018 VJ=100.00  +MOVJ EC00018 VJ=100.00
'Path S4515
SFTOF3D
MOVJ C00019 BC00019 VJ=100.00  +MOVJ EC00019 VJ=100.00
MOVL C00020 BC00020 V=800.0  +MOVJ EC00020 VJ=100.00
SMOVL C00021 BC00021 V=166.7  +MOVJ EC00021
SREFP 3 C00022 BC00022  +REFP EC00022
CALL JOB:SEARCH-R1-S13D
SET P033 P006
SFTON3D P033
SMOVL C00023 BC00023 V=250.0  +MOVJ EC00023
SMOVL C00024 BC00024 V=166.7  +MOVJ EC00024
SREFP 3 C00025 BC00025  +REFP EC00025
CALL JOB:SEARCH-R1-S13D
SET P033 P006
SFTON3D P033
SMOVL C00026 BC00026 V=166.7  +MOVJ EC00026
SMOVL C00027 BC00027 V=166.7  +MOVJ EC00027
SREFP 3 C00028 BC00028  +REFP EC00028
CALL JOB:SEARCH-R1-S13D
SET P033 P006
SFTON3D P033
SMOVL C00029 BC00029 V=166.7  +MOVJ EC00029
MOVL C00030 BC00030 V=1000.0  +MOVJ EC00030 VJ=100.00
'EndPath S4515
'Path S4516
SFTOF3D
MOVJ C00031 BC00031 VJ=100.00  +MOVJ EC00031 VJ=100.00
MOVL C00032 BC00032 V=800.0  +MOVJ EC00032 VJ=100.00
SMOVL C00033 BC00033 V=166.7  +MOVJ EC00033
SREFP 3 C00034 BC00034  +REFP EC00034
CALL JOB:SEARCH-R1-S13D
SET P032 P006
SFTON3D P032
SMOVL C00035 BC00035 V=166.7  +MOVJ EC00035
SMOVL C00036 BC00036 V=166.7  +MOVJ EC00036
SREFP 3 C00037 BC00037  +REFP EC00037
CALL JOB:SEARCH-R1-S13D
SET P032 P006
SFTON3D P032
SMOVL C00038 BC00038 V=166.7  +MOVJ EC00038
SMOVL C00039 BC00039 V=166.7  +MOVJ EC00039
SREFP 3 C00040 BC00040  +REFP EC00040
CALL JOB:SEARCH-R1-S13D
SET P032 P006
SFTON3D P032
SMOVL C00041 BC00041 V=166.7  +MOVJ EC00041
MOVL C00042 BC00042 V=1000.0  +MOVJ EC00042 VJ=100.00
'EndPath S4516
MOVJ C00043 BC00043 VJ=100.00  +MOVJ EC00043 VJ=100.00
MOVJ C00044 BC00044 VJ=100.00  +MOVJ EC00044 VJ=100.00
MOVL C00045 BC00045 V=800.0  +MOVJ EC00045 VJ=100.00
SMOVL C00046 BC00046 V=250.0  +MOVJ EC00046
SREFP 3 C00047 BC00047  +REFP EC00047
CALL JOB:SEARCH-R1-S13D
SET P099 P006
SFTON3D P099
SMOVL C00048 BC00048 V=166.7  +MOVJ EC00048
SMOVL C00049 BC00049 V=250.0  +MOVJ EC00049
SMOVL C00050 BC00050 V=166.7  +MOVJ EC00050
SREFP 3 C00051 BC00051  +REFP EC00051
CALL JOB:SEARCH-R1-S13D
SET P099 P006
SFTON3D P099
SMOVL C00052 BC00052 V=166.7  +MOVJ EC00052
SMOVL C00053 BC00053 V=800.0  +MOVJ EC00053
SFTOF3D
MOVJ C00054 BC00054 VJ=100.00  +MOVJ EC00054 VJ=100.00
'Path S4517
SFTOF3D
MOVJ C00055 BC00055 VJ=100.00  +MOVJ EC00055 VJ=100.00
'Path S4519
SFTOF3D
MOVJ C00056 BC00056 VJ=100.00  +MOVJ EC00056 VJ=100.00
MOVL C00057 BC00057 V=800.0  +MOVJ EC00057 VJ=100.00
SMOVL C00058 BC00058 V=166.7  +MOVJ EC00058
SREFP 3 C00059 BC00059  +REFP EC00059
CALL JOB:SEARCH-R1-S13D
SET P029 P006
SFTON3D P029
SMOVL C00060 BC00060 V=166.7  +MOVJ EC00060
SMOVL C00061 BC00061 V=166.7  +MOVJ EC00061
SREFP 3 C00062 BC00062  +REFP EC00062
CALL JOB:SEARCH-R1-S13D
SET P029 P006
SFTON3D P029
SMOVL C00063 BC00063 V=166.7  +MOVJ EC00063
SFTOF3D
MOVL C00064 BC00064 V=800.0  +MOVJ EC00064 VJ=100.00
MOVL C00065 BC00065 V=1000.0  +MOVJ EC00065 VJ=100.00
SMOVL C00066 BC00066 V=250.0  +MOVJ EC00066
SMOVL C00067 BC00067 V=250.0  +MOVJ EC00067
SREFP 3 C00068 BC00068  +REFP EC00068
CALL JOB:SEARCH-R1-S13D
SET P050 P006
SFTON3D P050
SMOVL C00069 BC00069 V=166.7  +MOVJ EC00069
SREFP 3 C00070 BC00070  +REFP EC00070
CALL JOB:SEARCH-R1-S13D
SET P050 P006
SFTON3D P050
SMOVL C00071 BC00071 V=166.7  +MOVJ EC00071
SMOVL C00072 BC00072 V=250.0  +MOVJ EC00072
SMOVL C00073 BC00073 V=250.0  +MOVJ EC00073
SREFP 3 C00074 BC00074  +REFP EC00074
CALL JOB:SEARCH-R1-S13D
SET P050 P006
SFTON3D P050
SMOVL C00075 BC00075 V=166.7  +MOVJ EC00075
SFTOF3D
SMOVL C00076 BC00076 V=666.7  +MOVJ EC00076
SMOVL C00077 BC00077 V=666.7  +MOVJ EC00077
SMOVL C00078 BC00078 V=250.0  +MOVJ EC00078
SMOVL C00079 BC00079 V=250.0  +MOVJ EC00079
SREFP 3 C00080 BC00080  +REFP EC00080
CALL JOB:SEARCH-R1-S13D
SET P051 P006
SFTON3D P051
SMOVL C00081 BC00081 V=166.7  +MOVJ EC00081
SMOVL C00082 BC00082 V=250.0  +MOVJ EC00082
SMOVL C00083 BC00083 V=133.3  +MOVJ EC00083
SREFP 3 C00084 BC00084  +REFP EC00084
CALL JOB:SEARCH-R1-S13D
SET P051 P006
SFTON3D P051
SMOVL C00085 BC00085 V=250.0  +MOVJ EC00085
SMOVL C00086 BC00086 V=500.0  +MOVJ EC00086
SMOVL C00087 BC00087 V=250.0  +MOVJ EC00087
SREFP 3 C00088 BC00088  +REFP EC00088
CALL JOB:SEARCH-R1-S13D
SET P051 P006
SFTON3D P051
SMOVL C00089 BC00089 V=166.7  +MOVJ EC00089
SFTOF3D
SMOVL C00090 BC00090 V=666.7  +MOVJ EC00090
'EndPath S4519
MOVJ C00091 BC00091 VJ=100.00  +MOVJ EC00091 VJ=100.00
'Path S4520
SFTOF3D
MOVJ C00092 BC00092 VJ=100.00  +MOVJ EC00092 VJ=100.00
MOVL C00093 BC00093 V=800.0  +MOVJ EC00093 VJ=100.00
SMOVL C00094 BC00094 V=133.3  +MOVJ EC00094
SREFP 3 C00095 BC00095  +REFP EC00095
CALL JOB:SEARCH-R1-S13D
SET P028 P006
SFTON3D P028
SMOVL C00096 BC00096 V=166.7  +MOVJ EC00096
SMOVL C00097 BC00097 V=166.7  +MOVJ EC00097
SREFP 3 C00098 BC00098  +REFP EC00098
CALL JOB:SEARCH-R1-S13D
SET P028 P006
SFTON3D P028
SMOVL C00099 BC00099 V=166.7  +MOVJ EC00099
MOVL C00100 BC00100 V=800.0  +MOVJ EC00100 VJ=100.00
MOVL C00101 BC00101 V=1000.0  +MOVJ EC00101 VJ=100.00
'EndPath S4520
'Path S4521
SFTOF3D
MOVJ C00102 BC00102 VJ=100.00  +MOVJ EC00102 VJ=100.00
MOVL C00103 BC00103 V=800.0  +MOVJ EC00103 VJ=100.00
SMOVL C00104 BC00104 V=166.7  +MOVJ EC00104
SREFP 3 C00105 BC00105  +REFP EC00105
CALL JOB:SEARCH-R1-S13D
SET P027 P006
SFTON3D P027
SMOVL C00106 BC00106 V=166.7  +MOVJ EC00106
SMOVL C00107 BC00107 V=166.7  +MOVJ EC00107
SREFP 3 C00108 BC00108  +REFP EC00108
CALL JOB:SEARCH-R1-S13D
SET P027 P006
SFTON3D P027
SMOVL C00109 BC00109 V=166.7  +MOVJ EC00109
MOVL C00110 BC00110 V=800.0  +MOVJ EC00110 VJ=100.00
MOVL C00111 BC00111 V=1000.0  +MOVJ EC00111 VJ=100.00
'EndPath S4521
MOVJ C00112 BC00112 VJ=100.00  +MOVJ EC00112 VJ=100.00
'Up
MOVJ C00113 BC00113 VJ=100.00  +MOVJ EC00113 VJ=100.00
MOVJ C00114 BC00114 VJ=100.00  +MOVJ EC00114 VJ=100.00
'Path S4522
SFTOF3D
MOVJ C00115 BC00115 VJ=100.00  +MOVJ EC00115 VJ=100.00
MOVL C00116 BC00116 V=800.0  +MOVJ EC00116 VJ=100.00
SMOVL C00117 BC00117 V=166.7  +MOVJ EC00117
SREFP 3 C00118 BC00118  +REFP EC00118
CALL JOB:SEARCH-R1-S13D
SET P026 P006
SFTON3D P026
SMOVL C00119 BC00119 V=166.7  +MOVJ EC00119
SREFP 3 C00120 BC00120  +REFP EC00120
CALL JOB:SEARCH-R1-S13D
SET P026 P006
SFTON3D P026
SMOVL C00121 BC00121 V=166.7  +MOVJ EC00121
MOVL C00122 BC00122 V=1000.0  +MOVJ EC00122 VJ=100.00
'EndPath S4522
'Path S4523
SFTOF3D
MOVJ C00123 BC00123 VJ=100.00  +MOVJ EC00123 VJ=100.00
MOVL C00124 BC00124 V=800.0  +MOVJ EC00124 VJ=100.00
SMOVL C00125 BC00125 V=166.7  +MOVJ EC00125
SREFP 3 C00126 BC00126  +REFP EC00126
CALL JOB:SEARCH-R1-S13D
SET P025 P006
SFTON3D P025
SMOVL C00127 BC00127 V=166.7  +MOVJ EC00127
SREFP 3 C00128 BC00128  +REFP EC00128
CALL JOB:SEARCH-R1-S13D
SET P025 P006
SFTON3D P025
SMOVL C00129 BC00129 V=166.7  +MOVJ EC00129
SMOVL C00130 BC00130 V=166.7  +MOVJ EC00130
SMOVL C00131 BC00131 V=166.7  +MOVJ EC00131
SREFP 3 C00132 BC00132  +REFP EC00132
CALL JOB:SEARCH-R1-S13D
SET P025 P006
SFTON3D P025
SMOVL C00133 BC00133 V=166.7  +MOVJ EC00133
MOVL C00134 BC00134 V=1000.0  +MOVJ EC00134 VJ=100.00
'EndPath S4523
'Path S4524
SFTOF3D
MOVJ C00135 BC00135 VJ=100.00  +MOVJ EC00135 VJ=100.00
MOVL C00136 BC00136 V=800.0  +MOVJ EC00136 VJ=100.00
SMOVL C00137 BC00137 V=166.7  +MOVJ EC00137
SREFP 3 C00138 BC00138  +REFP EC00138
CALL JOB:SEARCH-R1-S13D
SET P024 P006
SFTON3D P024
SMOVL C00139 BC00139 V=166.7  +MOVJ EC00139
SREFP 3 C00140 BC00140  +REFP EC00140
CALL JOB:SEARCH-R1-S13D
SET P024 P006
SFTON3D P024
SMOVL C00141 BC00141 V=166.7  +MOVJ EC00141
SMOVL C00142 BC00142 V=166.7  +MOVJ EC00142
SREFP 3 C00143 BC00143  +REFP EC00143
CALL JOB:SEARCH-R1-S13D
SET P024 P006
SFTON3D P024
SMOVL C00144 BC00144 V=166.7  +MOVJ EC00144
MOVL C00145 BC00145 V=1000.0  +MOVJ EC00145 VJ=100.00
'EndPath S4524
'Path S4525
SFTOF3D
MOVJ C00146 BC00146 VJ=100.00  +MOVJ EC00146 VJ=100.00
MOVL C00147 BC00147 V=800.0  +MOVJ EC00147 VJ=100.00
SMOVL C00148 BC00148 V=166.7  +MOVJ EC00148
SREFP 3 C00149 BC00149  +REFP EC00149
CALL JOB:SEARCH-R1-S13D
SET P023 P006
SFTON3D P023
SMOVL C00150 BC00150 V=166.7  +MOVJ EC00150
SREFP 3 C00151 BC00151  +REFP EC00151
CALL JOB:SEARCH-R1-S13D
SET P023 P006
SFTON3D P023
SMOVL C00152 BC00152 V=166.7  +MOVJ EC00152
SMOVL C00153 BC00153 V=166.7  +MOVJ EC00153
SREFP 3 C00154 BC00154  +REFP EC00154
CALL JOB:SEARCH-R1-S13D
SET P023 P006
SFTON3D P023
SMOVL C00155 BC00155 V=166.7  +MOVJ EC00155
MOVL C00156 BC00156 V=1000.0  +MOVJ EC00156 VJ=100.00
'EndPath S4525
'Path S4729
SFTOF3D
MOVJ C00157 BC00157 VJ=100.00  +MOVJ EC00157 VJ=100.00
MOVL C00158 BC00158 V=800.0  +MOVJ EC00158 VJ=100.00
SMOVL C00159 BC00159 V=166.7  +MOVJ EC00159
SREFP 3 C00160 BC00160  +REFP EC00160
CALL JOB:SEARCH-R1-S13D
SET P063 P006
SFTON3D P063
SMOVL C00161 BC00161 V=166.7  +MOVJ EC00161
SREFP 3 C00162 BC00162  +REFP EC00162
CALL JOB:SEARCH-R1-S13D
SET P063 P006
SFTON3D P063
SMOVL C00163 BC00163 V=166.7  +MOVJ EC00163
SMOVL C00164 BC00164 V=166.7  +MOVJ EC00164
SREFP 3 C00165 BC00165  +REFP EC00165
CALL JOB:SEARCH-R1-S13D
SET P063 P006
SFTON3D P063
SMOVL C00166 BC00166 V=166.7  +MOVJ EC00166
MOVL C00167 BC00167 V=1000.0  +MOVJ EC00167 VJ=100.00
'EndPath S4729
'Path S4526
SFTOF3D
MOVJ C00168 BC00168 VJ=100.00  +MOVJ EC00168 VJ=100.00
MOVL C00169 BC00169 V=800.0  +MOVJ EC00169 VJ=100.00
SMOVL C00170 BC00170 V=166.7  +MOVJ EC00170
SREFP 3 C00171 BC00171  +REFP EC00171
CALL JOB:SEARCH-R1-S13D
SET P022 P006
SFTON3D P022
SMOVL C00172 BC00172 V=166.7  +MOVJ EC00172
SREFP 3 C00173 BC00173  +REFP EC00173
CALL JOB:SEARCH-R1-S13D
SET P022 P006
SFTON3D P022
SMOVL C00174 BC00174 V=166.7  +MOVJ EC00174
SREFP 3 C00175 BC00175  +REFP EC00175
CALL JOB:SEARCH-R1-S13D
SET P022 P006
SFTON3D P022
SMOVL C00176 BC00176 V=166.7  +MOVJ EC00176
MOVL C00177 BC00177 V=1000.0  +MOVJ EC00177 VJ=100.00
'EndPath S4526
'Path S4527
SFTOF3D
MOVJ C00178 BC00178 VJ=100.00  +MOVJ EC00178 VJ=100.00
MOVL C00179 BC00179 V=800.0  +MOVJ EC00179 VJ=100.00
SMOVL C00180 BC00180 V=166.7  +MOVJ EC00180
SREFP 3 C00181 BC00181  +REFP EC00181
CALL JOB:SEARCH-R1-S13D
SET P021 P006
SFTON3D P021
SMOVL C00182 BC00182 V=166.7  +MOVJ EC00182
SREFP 3 C00183 BC00183  +REFP EC00183
CALL JOB:SEARCH-R1-S13D
SET P021 P006
SFTON3D P021
SMOVL C00184 BC00184 V=250.0  +MOVJ EC00184
SMOVL C00185 BC00185 V=166.7  +MOVJ EC00185
SREFP 3 C00186 BC00186  +REFP EC00186
CALL JOB:SEARCH-R1-S13D
SET P021 P006
SFTON3D P021
SMOVL C00187 BC00187 V=166.7  +MOVJ EC00187
MOVL C00188 BC00188 V=1000.0  +MOVJ EC00188 VJ=100.00
'EndPath S4527
MOVJ C00189 BC00189 VJ=100.00  +MOVJ EC00189 VJ=100.00
'Path W4730
SFTOF3D
SFTON3D P024
MOVJ C00190 BC00190 VJ=100.00  +MOVJ EC00190 VJ=100.00
SMOVL C00191 BC00191 V=800.0  +MOVJ EC00191
SMOVL C00192 BC00192 V=150.0 PL=0  +MOVJ EC00192
MACRO1 MJ#(0) ARGF14
ARCON
SMOVL C00193 BC00193 V=10.0  +MOVJ EC00193
SMOVL C00194 BC00194 V=11.7  +MOVJ EC00194
ARCOF
SMOVL C00195 BC00195 V=800.0  +MOVJ EC00195
SMOVL C00196 BC00196 V=1000.0  +MOVJ EC00196
SFTOF3D
'EndPath W4730
MOVJ C00197 BC00197 VJ=100.00  +MOVJ EC00197 VJ=100.00
'Path W4731
SFTOF3D
SFTON3D P063
MOVJ C00198 BC00198 VJ=100.00  +MOVJ EC00198 VJ=100.00
SMOVL C00199 BC00199 V=800.0  +MOVJ EC00199
SMOVL C00200 BC00200 V=150.0 PL=0  +MOVJ EC00200
MACRO1 MJ#(0) ARGF9
ARCON
SMOVL C00201 BC00201 V=10.0  +MOVJ EC00201
SMOVL C00202 BC00202 V=10.0  +MOVJ EC00202
ARCOF
SMOVL C00203 BC00203 V=800.0  +MOVJ EC00203
SMOVL C00204 BC00204 V=1000.0  +MOVJ EC00204
SFTOF3D
'EndPath W4731
'Path W4528
SFTOF3D
SFTON3D P021
MOVJ C00205 BC00205 VJ=100.00  +MOVJ EC00205 VJ=100.00
SMOVL C00206 BC00206 V=800.0  +MOVJ EC00206
SMOVL C00207 BC00207 V=166.7 PL=0  +MOVJ EC00207
MACRO1 MJ#(0) ARGF21
ARCON
SMOVL C00208 BC00208 V=10.8  +MOVJ EC00208
SFTON3D P022
SMOVL C00209 BC00209 V=10.8  +MOVJ EC00209
SMOVL C00210 BC00210 V=10.8  +MOVJ EC00210
ARCOF
SMOVL C00211 BC00211 V=800.0  +MOVJ EC00211
SMOVL C00212 BC00212 V=1000.0  +MOVJ EC00212
SFTOF3D
'EndPath W4528
'Path W4529
SFTOF3D
SFTON3D P022
MOVJ C00213 BC00213 VJ=100.00  +MOVJ EC00213 VJ=100.00
SMOVL C00214 BC00214 V=800.0  +MOVJ EC00214
SMOVL C00215 BC00215 V=166.7 PL=0  +MOVJ EC00215
ARCON
SMOVL C00216 BC00216 V=10.8  +MOVJ EC00216
ARCOF
SMOVL C00217 BC00217 V=800.0  +MOVJ EC00217
SMOVL C00218 BC00218 V=1000.0  +MOVJ EC00218
SFTOF3D
'EndPath W4529
'Path W4530
SFTOF3D
SFTON3D P023
MOVJ C00219 BC00219 VJ=100.00  +MOVJ EC00219 VJ=100.00
SMOVL C00220 BC00220 V=800.0  +MOVJ EC00220
SMOVL C00221 BC00221 V=166.7 PL=0  +MOVJ EC00221
ARCON
SWVON WEV#(60)
SMOVL C00222 BC00222 V=7.5  +MOVJ EC00222
SFTON3D P024
SMOVL C00223 BC00223 V=7.5  +MOVJ EC00223
SMOVL C00224 BC00224 V=7.5  +MOVJ EC00224
ARCOF
SWVOF
SMOVL C00225 BC00225 V=800.0  +MOVJ EC00225
SMOVL C00226 BC00226 V=1000.0  +MOVJ EC00226
SFTOF3D
'EndPath W4530
'Path W4531
SFTOF3D
SFTON3D P025
MOVJ C00227 BC00227 VJ=100.00  +MOVJ EC00227 VJ=100.00
SMOVL C00228 BC00228 V=800.0  +MOVJ EC00228
SMOVL C00229 BC00229 V=166.7 PL=0  +MOVJ EC00229
ARCON
SMOVL C00230 BC00230 V=10.8  +MOVJ EC00230
SFTON3D P026
SMOVL C00231 BC00231 V=10.8  +MOVJ EC00231
SMOVL C00232 BC00232 V=10.8  +MOVJ EC00232
ARCOF
SMOVL C00233 BC00233 V=800.0  +MOVJ EC00233
SMOVL C00234 BC00234 V=1000.0  +MOVJ EC00234
SFTOF3D
'EndPath W4531
'Down
MOVJ C00235 BC00235 VJ=100.00  +MOVJ EC00235 VJ=100.00
MOVJ C00236 BC00236 VJ=100.00  +MOVJ EC00236 VJ=100.00
MOVJ C00237 BC00237 VJ=100.00  +MOVJ EC00237 VJ=100.00
MOVJ C00238 BC00238 VJ=100.00  +MOVJ EC00238 VJ=100.00
'Path W4532
SFTOF3D
MOVJ C00239 BC00239 VJ=100.00  +MOVJ EC00239 VJ=100.00
MOVJ C00240 BC00240 VJ=100.00  +MOVJ EC00240 VJ=100.00
'Path W4534
SFTOF3D
SFTON3D P033
MOVJ C00241 BC00241 VJ=100.00  +MOVJ EC00241 VJ=100.00
SMOVL C00242 BC00242 V=800.0  +MOVJ EC00242
SMOVL C00243 BC00243 V=166.7 PL=0  +MOVJ EC00243
MACRO1 MJ#(0) ARGF14
ARCON
SMOVL C00244 BC00244 V=10.0  +MOVJ EC00244
SMOVL C00245 BC00245 V=10.0  +MOVJ EC00245
SMOVL C00246 BC00246 V=10.0  +MOVJ EC00246
ARCOF
SMOVL C00247 BC00247 V=800.0  +MOVJ EC00247
SMOVL C00248 BC00248 V=166.7  +MOVJ EC00248
SMOVL C00249 BC00249 V=166.7  +MOVJ EC00249
ARCON
SMOVL C00250 BC00250 V=13.3  +MOVJ EC00250
SMOVL C00251 BC00251 V=13.3  +MOVJ EC00251
ARCOF
SMOVL C00252 BC00252 V=166.7  +MOVJ EC00252
SMOVL C00253 BC00253 V=500.0  +MOVJ EC00253
SMOVL C00254 BC00254 V=133.3  +MOVJ EC00254
ARCON
SMOVL C00255 BC00255 V=13.3  +MOVJ EC00255
SMOVL C00256 BC00256 V=13.3  +MOVJ EC00256
ARCOF
SMOVL C00257 BC00257 V=250.0  +MOVJ EC00257
SMOVL C00258 BC00258 V=1000.0  +MOVJ EC00258
SFTOF3D
'EndPath W4534
'Path W4535
SFTOF3D
SFTON3D P032
MOVJ C00259 BC00259 VJ=100.00  +MOVJ EC00259 VJ=100.00
SMOVL C00260 BC00260 V=800.0  +MOVJ EC00260
SMOVL C00261 BC00261 V=166.7 PL=0  +MOVJ EC00261
ARCON
SMOVL C00262 BC00262 V=10.0  +MOVJ EC00262
SMOVL C00263 BC00263 V=10.0  +MOVJ EC00263
SMOVL C00264 BC00264 V=10.0  +MOVJ EC00264
ARCOF
SMOVL C00265 BC00265 V=800.0  +MOVJ EC00265
SMOVL C00266 BC00266 V=250.0  +MOVJ EC00266
SMOVL C00267 BC00267 V=166.7  +MOVJ EC00267
ARCON
SMOVL C00268 BC00268 V=10.8  +MOVJ EC00268
ARCOF
SMOVL C00269 BC00269 V=250.0  +MOVJ EC00269
SMOVL C00270 BC00270 V=1000.0  +MOVJ EC00270
SFTOF3D
'EndPath W4535
'Path W4536
SFTOF3D
SFTON3D P032
MOVJ C00271 BC00271 VJ=100.00  +MOVJ EC00271 VJ=100.00
SFTOF3D
'EndPath W4536
MOVJ C00272 BC00272 VJ=100.00  +MOVJ EC00272 VJ=100.00
'Path W4537
SFTOF3D
SFTON3D P027
MOVJ C00273 BC00273 VJ=100.00  +MOVJ EC00273 VJ=100.00
SMOVL C00274 BC00274 V=800.0  +MOVJ EC00274
SMOVL C00275 BC00275 V=150.0 PL=0  +MOVJ EC00275
MACRO1 MJ#(0) ARGF9
ARCON
SMOVL C00276 BC00276 V=10.8  +MOVJ EC00276
SMOVL C00277 BC00277 V=10.8  +MOVJ EC00277
ARCOF
SMOVL C00278 BC00278 V=800.0  +MOVJ EC00278
SMOVL C00279 BC00279 V=1000.0  +MOVJ EC00279
SFTOF3D
'EndPath W4537
'Path W4538
SFTOF3D
SFTON3D P027
SMOVL C00280 BC00280 V=1000.0  +MOVJ EC00280
SMOVL C00281 BC00281 V=150.0 PL=0  +MOVJ EC00281
ARCON
SMOVL C00282 BC00282 V=10.8  +MOVJ EC00282
ARCOF
SMOVL C00283 BC00283 V=800.0  +MOVJ EC00283
SFTOF3D
'EndPath W4538
'Path W4539
SFTOF3D
SFTON3D P028
SMOVL C00284 BC00284 V=1000.0  +MOVJ EC00284
SMOVL C00285 BC00285 V=150.0 PL=0  +MOVJ EC00285
ARCON
SMOVL C00286 BC00286 V=10.8  +MOVJ EC00286
ARCOF
SMOVL C00287 BC00287 V=800.0  +MOVJ EC00287
SFTOF3D
'EndPath W4539
'Path W4540
SFTOF3D
SFTON3D P028
SMOVL C00288 BC00288 V=1000.0  +MOVJ EC00288
SMOVL C00289 BC00289 V=150.0 PL=0  +MOVJ EC00289
ARCON
SMOVL C00290 BC00290 V=10.8  +MOVJ EC00290
SMOVL C00291 BC00291 V=10.8  +MOVJ EC00291
ARCOF
SMOVL C00292 BC00292 V=800.0  +MOVJ EC00292
SMOVL C00293 BC00293 V=1000.0  +MOVJ EC00293
SFTOF3D
'EndPath W4540
MOVJ C00294 BC00294 VJ=100.00  +MOVJ EC00294 VJ=100.00
MOVJ C00295 BC00295 VJ=100.00  +MOVJ EC00295 VJ=100.00
SMOVL C00296 BC00296 V=666.7  +MOVJ EC00296
MACRO1 MJ#(0) ARGF14
SFTON3D P051
SMOVL C00297 BC00297 V=166.7  +MOVJ EC00297
ARCON
SMOVL C00298 BC00298 V=10.8  +MOVJ EC00298
ARCOF
SMOVL C00299 BC00299 V=133.3  +MOVJ EC00299
SMOVL C00300 BC00300 V=133.3  +MOVJ EC00300
ARCON
SMOVL C00301 BC00301 V=6.7  +MOVJ EC00301
ARCOF
SMOVL C00302 BC00302 V=133.3  +MOVJ EC00302
SMOVL C00303 BC00303 V=250.0  +MOVJ EC00303
MACRO1 MJ#(0) ARGF9
SMOVL C00304 BC00304 V=133.3  +MOVJ EC00304
ARCON
SMOVL C00305 BC00305 V=8.3  +MOVJ EC00305
ARCOF
SMOVL C00306 BC00306 V=250.0  +MOVJ EC00306
SMOVL C00307 BC00307 V=250.0  +MOVJ EC00307
MACRO1 MJ#(0) ARGF14
SMOVL C00308 BC00308 V=166.7  +MOVJ EC00308
ARCON
SMOVL C00309 BC00309 V=10.8  +MOVJ EC00309
ARCOF
SMOVL C00310 BC00310 V=166.7  +MOVJ EC00310
SFTON3D P050
SMOVL C00311 BC00311 V=166.7  +MOVJ EC00311
ARCON
SMOVL C00312 BC00312 V=10.8  +MOVJ EC00312
ARCOF
SMOVL C00313 BC00313 V=166.7  +MOVJ EC00313
ARCON
SMOVL C00314 BC00314 V=11.7  +MOVJ EC00314
SMOVL C00315 BC00315 V=11.7  +MOVJ EC00315
ARCOF
SMOVL C00316 BC00316 V=166.7  +MOVJ EC00316
SFTOF3D
MOVJ C00317 BC00317 VJ=100.00  +MOVJ EC00317 VJ=100.00
'Path W4541
SFTOF3D
SFTON3D P029
MOVJ C00318 BC00318 VJ=100.00  +MOVJ EC00318 VJ=100.00
SMOVL C00319 BC00319 V=800.0  +MOVJ EC00319
MACRO1 MJ#(0) ARGF9
SMOVL C00320 BC00320 V=150.0 PL=0  +MOVJ EC00320
ARCON
SMOVL C00321 BC00321 V=10.8  +MOVJ EC00321
ARCOF
SMOVL C00322 BC00322 V=800.0  +MOVJ EC00322
SMOVL C00323 BC00323 V=1000.0  +MOVJ EC00323
SFTOF3D
'EndPath W4541
'Path W4542
SFTOF3D
SFTON3D P029
MOVJ C00324 BC00324 VJ=100.00  +MOVJ EC00324 VJ=100.00
SMOVL C00325 BC00325 V=800.0  +MOVJ EC00325
SMOVL C00326 BC00326 V=150.0 PL=0  +MOVJ EC00326
ARCON
SMOVL C00327 BC00327 V=10.8  +MOVJ EC00327
ARCOF
SMOVL C00328 BC00328 V=800.0  +MOVJ EC00328
SMOVL C00329 BC00329 V=1000.0  +MOVJ EC00329
SFTOF3D
'EndPath W4542
MOVJ C00330 BC00330 VJ=100.00  +MOVJ EC00330 VJ=100.00
MOVJ C00331 BC00331 VJ=100.00  +MOVJ EC00331 VJ=100.00
MOVJ C00332 BC00332 VJ=100.00  +MOVJ EC00332 VJ=100.00
MOVJ C00333 BC00333 VJ=100.00  +MOVJ EC00333 VJ=100.00
SFTON3D P099
SMOVL C00334 BC00334 V=166.7  +MOVJ EC00334
ARCON
SMOVL C00335 BC00335 V=10.8  +MOVJ EC00335
ARCOF
SFTOF3D
SMOVL C00336 BC00336 V=166.7  +MOVJ EC00336
MOVJ C00337 BC00337 VJ=100.00  +MOVJ EC00337 VJ=100.00
MOVJ C00338 BC00338 VJ=100.00  +MOVJ EC00338 VJ=100.00
MOVJ C00339 BC00339 VJ=100.00  +MOVJ EC00339 VJ=100.00
MOVJ C00340 BC00340 VJ=100.00  +MOVJ EC00340 VJ=100.00
SFTON3D P050
SMOVL C00341 BC00341 V=166.7  +MOVJ EC00341
ARCON
SMOVL C00342 BC00342 V=11.7  +MOVJ EC00342
ARCOF
SMOVL C00343 BC00343 V=133.3  +MOVJ EC00343
SMOVL C00344 BC00344 V=133.3  +MOVJ EC00344
SMOVL C00345 BC00345 V=133.3  +MOVJ EC00345
ARCON
SMOVL C00346 BC00346 V=10.8  +MOVJ EC00346
ARCOF
SMOVL C00347 BC00347 V=416.7  +MOVJ EC00347
SFTOF3D
MOVJ C00348 BC00348 VJ=100.00  +MOVJ EC00348 VJ=100.00
MOVJ C00349 BC00349 VJ=100.00  +MOVJ EC00349 VJ=100.00
MOVJ C00350 BC00350 VJ=100.00  +MOVJ EC00350 VJ=100.00
SFTON3D P032
SMOVL C00351 BC00351 V=133.3  +MOVJ EC00351
ARCON
SMOVL C00352 BC00352 V=13.3  +MOVJ EC00352
SMOVL C00353 BC00353 V=13.3  +MOVJ EC00353
SMOVL C00354 BC00354 V=13.3  +MOVJ EC00354
ARCOF
SMOVL C00355 BC00355 V=250.0  +MOVJ EC00355
SMOVL C00356 BC00356 V=666.7  +MOVJ EC00356
MOVJ C00357 BC00357 VJ=100.00  +MOVJ EC00357 VJ=100.00
MOVJ C00358 BC00358 VJ=100.00  +MOVJ EC00358 VJ=100.00
'Path W4543
SFTOF3D
SFTON3D P034
MOVJ C00359 BC00359 VJ=100.00  +MOVJ EC00359 VJ=100.00
SMOVL C00360 BC00360 V=800.0  +MOVJ EC00360
SMOVL C00361 BC00361 V=150.0 PL=0  +MOVJ EC00361
MACRO1 MJ#(0) ARGF14
ARCON
SMOVL C00362 BC00362 V=10.8  +MOVJ EC00362
SMOVL C00363 BC00363 V=10.8  +MOVJ EC00363
ARCOF
SMOVL C00364 BC00364 V=800.0  +MOVJ EC00364
SMOVL C00365 BC00365 V=333.3  +MOVJ EC00365
SMOVL C00366 BC00366 V=133.3  +MOVJ EC00366
ARCON
SMOVL C00367 BC00367 V=10.8  +MOVJ EC00367
SMOVL C00368 BC00368 V=10.8  +MOVJ EC00368
ARCOF
SMOVL C00369 BC00369 V=166.7  +MOVJ EC00369
SMOVL C00370 BC00370 V=166.7  +MOVJ EC00370
SMOVL C00371 BC00371 V=166.7  +MOVJ EC00371
SMOVL C00372 BC00372 V=166.7  +MOVJ EC00372
ARCON
SMOVL C00373 BC00373 V=10.8  +MOVJ EC00373
ARCOF
SMOVL C00374 BC00374 V=166.7  +MOVJ EC00374
SMOVL C00375 BC00375 V=166.7  +MOVJ EC00375
SFTOF3D
'EndPath W4543
MOVJ C00376 BC00376 VJ=100.00  +MOVJ EC00376 VJ=100.00
MOVJ C00377 BC00377 VJ=100.00  +MOVJ EC00377 VJ=100.00
END
